TYPE ST_PDxx_PredefinedErrorField :
STRUCT
	nErrorNumber	: USINT;
	stErrorClass	: ST_PDxx_ErrorRegister;
	nErrorCode		: UINT;
END_STRUCT
END_TYPE

(* stored: Version 1.1.0.1, ProductVersion 3.1.4024.15
   DUT ST_PDxx_PredefinedErrorField: Id {6f8fb9bc-1955-409b-908a-0d47258a147a} *)
